ABB RAPID module: Module1.mod

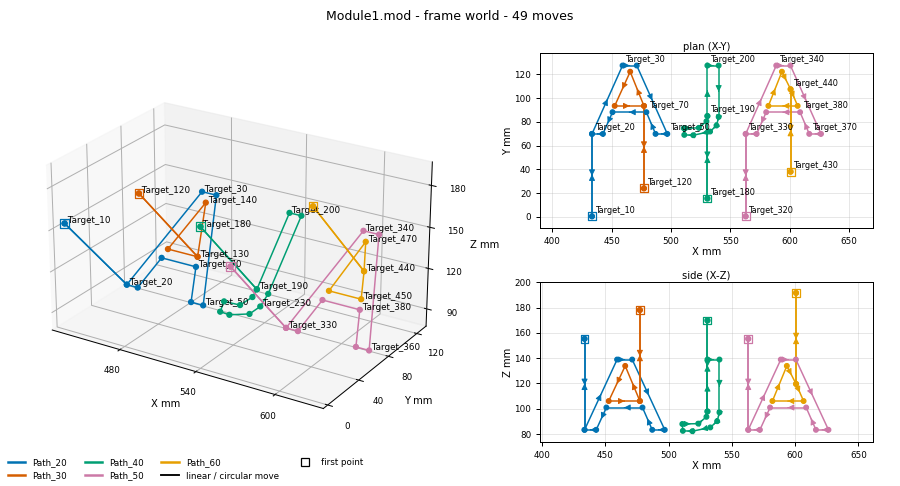
[picture p0: tool path of Module1.mod in frame world, 49 of 55 moves have a stored position in this frame; points joined in program order, loops and branches not executed]
MODULE Module1
        CONST robtarget Target_10:=[[-33.51704764,187.401145356,100.000301826],[0.00000002,-0.58897389,0.808152063,0.000000028],[-1,1,-1,1],[9E+09,9E+09,9E+09,9E+09,9E+09,9E+09]];
    CONST robtarget Target_20:=[[-33.51704764,187.401152167,0.000301826],[0.00000002,-0.58897389,0.808152063,0.000000028],[0,1,-1,1],[9E+09,9E+09,9E+09,9E+09,9E+09,9E+09]];
    CONST robtarget Target_30:=[[-59.250836036,107.401152167,0.000296377],[0.00000002,-0.58897389,0.808152063,0.000000028],[0,1,-1,1],[9E+09,9E+09,9E+09,9E+09,9E+09,9E+09]];
    CONST robtarget Target_40:=[[-71.196228528,107.401152167,0.000296377],[0.00000002,-0.58897389,0.808152063,0.000000028],[0,1,-1,1],[9E+09,9E+09,9E+09,9E+09,9E+09,9E+09]];
    CONST robtarget Target_50:=[[-96.930016924,187.401152167,0.000301826],[0.000000025,0.720360186,-0.693600175,-0.000000024],[0,1,-1,1],[9E+09,9E+09,9E+09,9E+09,9E+09,9E+09]];
    CONST robtarget Target_60:=[[-87.032406002,187.401152167,0.000301826],[0.00000002,-0.58897389,0.808152063,0.000000028],[0,1,-1,1],[9E+09,9E+09,9E+09,9E+09,9E+09,9E+09]];
    CONST robtarget Target_70:=[[-79.319095422,162.0086607,0.000300096],[0.00000002,-0.58897389,0.808152063,0.000000028],[0,1,-1,1],[9E+09,9E+09,9E+09,9E+09,9E+09,9E+09]];
    CONST robtarget Target_80:=[[-50.786672214,162.0086607,0.000300096],[0.00000002,-0.58897389,0.808152063,0.000000028],[0,1,-1,1],[9E+09,9E+09,9E+09,9E+09,9E+09,9E+09]];
    CONST robtarget Target_90:=[[-42.732064705,187.401152167,0.000301826],[0.00000002,-0.58897389,0.808152063,0.000000028],[0,1,-1,1],[9E+09,9E+09,9E+09,9E+09,9E+09,9E+09]];
    CONST robtarget Target_100:=[[-33.51704764,187.401152167,0.000301826],[0.00000002,-0.58897389,0.808152063,0.000000028],[0,1,-1,1],[9E+09,9E+09,9E+09,9E+09,9E+09,9E+09]];
    CONST robtarget Target_110:=[[-33.51704764,187.401145356,100.000301826],[0.00000002,-0.58897389,0.808152063,0.000000028],[-1,1,-1,1],[9E+09,9E+09,9E+09,9E+09,9E+09,9E+09]];
    CONST robtarget Target_120:=[[-77.271313852,154.636640237,100.000299594],[0.000000027,0.803729665,-0.594994644,-0.000000021],[0,1,-1,1],[9E+09,9E+09,9E+09,9E+09,9E+09,9E+09]];
    CONST robtarget Target_130:=[[-77.271313852,154.636647047,0.000299594],[-0.000000027,0.803729665,-0.594994644,-0.000000021],[0,1,-1,1],[9E+09,9E+09,9E+09,9E+09,9E+09,9E+09]];
    CONST robtarget Target_140:=[[-65.667218289,114.636647047,0.00029687],[-0.000000027,0.803729665,-0.594994644,-0.000000021],[0,1,-1,1],[9E+09,9E+09,9E+09,9E+09,9E+09,9E+09]];
    CONST robtarget Target_150:=[[-52.629675627,154.636647047,0.000299594],[-0.000000027,0.803729665,-0.594994644,-0.000000021],[0,1,-1,1],[9E+09,9E+09,9E+09,9E+09,9E+09,9E+09]];
    CONST robtarget Target_160:=[[-77.271313852,154.636647047,0.000299594],[-0.000000027,0.803729665,-0.594994644,-0.000000021],[0,1,-1,1],[9E+09,9E+09,9E+09,9E+09,9E+09,9E+09]];
    CONST robtarget Target_170:=[[-77.271313852,154.636640237,100.000299594],[-0.000000027,0.803729665,-0.594994644,-0.000000021],[0,1,-1,1],[9E+09,9E+09,9E+09,9E+09,9E+09,9E+09]];
    CONST robtarget Target_180:=[[-130.684278975,166.513773343,100.000300403],[-0.000000024,0.819152044,-0.573576437,-0.000000024],[0,1,-1,1],[9E+09,9E+09,9E+09,9E+09,9E+09,9E+09]];
    CONST robtarget Target_190:=[[-130.684278975,166.513780154,0.000300403],[0.000000024,-0.707106781,0.707106781,0.000000024],[0,1,-1,1],[9E+09,9E+09,9E+09,9E+09,9E+09,9E+09]];
    CONST robtarget Target_200:=[[-130.684278975,107.401152167,0.000296377],[0.000000024,-0.707106781,0.707106781,0.000000024],[0,1,-1,1],[9E+09,9E+09,9E+09,9E+09,9E+09,9E+09]];
    CONST robtarget Target_210:=[[-140.172333582,107.401152167,0.000296377],[0.000000024,-0.707106781,0.707106781,0.000000024],[0,1,-1,1],[9E+09,9E+09,9E+09,9E+09,9E+09,9E+09]];
    CONST robtarget Target_220:=[[-140.172333582,167.537670939,0.000300473],[0.000000024,0.819152044,-0.573576437,-0.000000024],[0,1,-1,1],[9E+09,9E+09,9E+09,9E+09,9E+09,9E+09]];
    CONST robtarget Target_230:=[[-138.363459862,177.588865478,0.000301158],[0.000000024,0.819152044,-0.573576437,-0.000000024],[0,1,-1,1],[9E+09,9E+09,9E+09,9E+09,9E+09,9E+09]];
    CONST robtarget Target_240:=[[-132.936838702,184.67077674,0.00030164],[0.000000024,0.819152044,-0.573576437,-0.000000024],[0,1,-1,1],[9E+09,9E+09,9E+09,9E+09,9E+09,9E+09]];
    CONST robtarget Target_250:=[[-118.807145869,188.971118037,0.000301932],[0.000000024,-0.707106781,0.707106781,0.000000024],[0,1,-1,1],[9E+09,9E+09,9E+09,9E+09,9E+09,9E+09]];
    CONST robtarget Target_260:=[[-111.23035406,188.561561724,0.000301905],[0.000000024,-0.707106781,0.707106781,0.000000024],[0,1,-1,1],[9E+09,9E+09,9E+09,9E+09,9E+09,9E+09]];
    CONST robtarget Target_270:=[[-110.820797746,180.779991758,0.000301375],[0.000000024,-0.707106781,0.707106781,0.000000024],[0,1,-1,1],[9E+09,9E+09,9E+09,9E+09,9E+09,9E+09]];
    CONST robtarget Target_280:=[[-123.482913787,180.353370597,0.000301346],[0.000000024,-0.707106781,0.707106781,0.000000024],[0,1,-1,1],[9E+09,9E+09,9E+09,9E+09,9E+09,9E+09]];
    CONST robtarget Target_290:=[[-129.882231193,172.605930324,0.000300819],[0.000000024,-0.707106781,0.707106781,0.000000024],[0,1,-1,1],[9E+09,9E+09,9E+09,9E+09,9E+09,9E+09]];
    CONST robtarget Target_300:=[[-130.684278975,166.513780154,0.000300403],[0.000000024,-0.707106781,0.707106781,0.000000024],[0,1,-1,1],[9E+09,9E+09,9E+09,9E+09,9E+09,9E+09]];
    CONST robtarget Target_310:=[[-130.684278975,166.513773343,100.000300403],[0.000000024,0.819152044,-0.573576437,-0.000000024],[0,1,-1,1],[9E+09,9E+09,9E+09,9E+09,9E+09,9E+09]];
    CONST robtarget Target_320:=[[-162.936835762,187.401145356,100.000301826],[-0.000000002,0.707106782,-0.70710678,-0.000000035],[-1,1,-1,1],[9E+09,9E+09,9E+09,9E+09,9E+09,9E+09]];
    CONST robtarget Target_330:=[[-162.936835762,187.401152167,0.000301826],[0.000000002,0.707106782,-0.70710678,-0.000000035],[0,1,-1,1],[9E+09,9E+09,9E+09,9E+09,9E+09,9E+09]];
    CONST robtarget Target_340:=[[-188.670624158,107.401152167,0.000296377],[0.000000002,0.707106782,-0.70710678,-0.000000035],[0,1,-1,1],[9E+09,9E+09,9E+09,9E+09,9E+09,9E+09]];
    CONST robtarget Target_350:=[[-200.61601665,107.401152167,0.000296377],[0.000000002,0.707106782,-0.70710678,-0.000000035],[0,1,-1,1],[9E+09,9E+09,9E+09,9E+09,9E+09,9E+09]];
    CONST robtarget Target_360:=[[-226.349805046,187.401152167,0.000301826],[0.000000002,0.707106782,-0.70710678,-0.000000035],[0,1,-1,1],[9E+09,9E+09,9E+09,9E+09,9E+09,9E+09]];
    CONST robtarget Target_370:=[[-216.452194124,187.401152167,0.000301826],[0.000000002,0.707106782,-0.70710678,-0.000000035],[0,1,-1,1],[9E+09,9E+09,9E+09,9E+09,9E+09,9E+09]];
    CONST robtarget Target_380:=[[-208.738883544,162.0086607,0.000300096],[0.000000002,0.707106782,-0.70710678,-0.000000035],[0,1,-1,1],[9E+09,9E+09,9E+09,9E+09,9E+09,9E+09]];
    CONST robtarget Target_390:=[[-180.206460336,162.0086607,0.000300096],[0.000000002,0.707106782,-0.70710678,-0.000000035],[0,1,-1,1],[9E+09,9E+09,9E+09,9E+09,9E+09,9E+09]];
    CONST robtarget Target_400:=[[-172.151852827,187.401152167,0.000301826],[0.000000002,0.707106782,-0.70710678,-0.000000035],[0,1,-1,1],[9E+09,9E+09,9E+09,9E+09,9E+09,9E+09]];
    CONST robtarget Target_410:=[[-162.936835762,187.401152167,0.000301826],[0.000000002,0.707106782,-0.70710678,-0.000000035],[0,1,-1,1],[9E+09,9E+09,9E+09,9E+09,9E+09,9E+09]];
    CONST robtarget Target_420:=[[-162.936835762,187.401145356,100.000301826],[0.000000002,0.707106782,-0.70710678,-0.000000035],[-1,1,-1,1],[9E+09,9E+09,9E+09,9E+09,9E+09,9E+09]];
    CONST robtarget Target_430:=[[-200.752535421,135.182715322,100.00029827],[0.000000021,-0.61876536,0.785575858,0.000000027],[0,1,-1,1],[9E+09,9E+09,9E+09,9E+09,9E+09,9E+09]];
    CONST robtarget Target_440:=[[-200.752535421,135.182722133,0.000298269],[0.000000021,-0.61876536,0.785575858,0.000000027],[0,1,-1,1],[9E+09,9E+09,9E+09,9E+09,9E+09,9E+09]];
    CONST robtarget Target_450:=[[-206.691101974,154.636647047,0.000299594],[0.000000021,-0.61876536,0.785575858,0.000000027],[0,1,-1,1],[9E+09,9E+09,9E+09,9E+09,9E+09,9E+09]];
    CONST robtarget Target_460:=[[-182.049463749,154.636647047,0.000299594],[0.000000021,-0.61876536,0.785575858,0.000000027],[0,1,-1,1],[9E+09,9E+09,9E+09,9E+09,9E+09,9E+09]];
    CONST robtarget Target_470:=[[-193.448781155,114.636647047,0.00029687],[0.000000021,-0.61876536,0.785575858,0.000000027],[0,1,-1,1],[9E+09,9E+09,9E+09,9E+09,9E+09,9E+09]];
    CONST robtarget Target_480:=[[-200.752535421,135.182722133,0.000298269],[0.000000021,-0.61876536,0.785575858,0.000000027],[0,1,-1,1],[9E+09,9E+09,9E+09,9E+09,9E+09,9E+09]];
    CONST robtarget Target_490:=[[-200.752535421,135.182715322,100.00029827],[0.000000021,-0.61876536,0.785575858,0.000000027],[0,1,-1,1],[9E+09,9E+09,9E+09,9E+09,9E+09,9E+09]];
    CONST jointtarget HomeP:=[[0,0,0,0,0,0],[9E+09,9E+09,9E+09,9E+09,9E+09,9E+09]];
    CONST jointtarget JointTarget_1:=[[0,20,-20,40,-20,-20],[9E+09,9E+09,9E+09,9E+09,9E+09,9E+09]];
    CONST jointtarget JointTarget_2:=[[0,50,-40,70,-50,-50],[9E+09,9E+09,9E+09,9E+09,9E+09,9E+09]];
!***********************************************************
    !
    ! Módulo:  Module1
    !
    ! Descripción:
    !   <Introduzca la descripción aquí>
    !
    ! Autor: equip
    !
    ! Versión: 1.0
    !
    !***********************************************************


    !***********************************************************
    !
    ! Procedimiento Main
    !
    !   Este es el punto de entrada de su programa
    !
    !***********************************************************
    PROC main()
        Security;
        Path_20;
        Path_30;
        Path_40;
        Path_50;
        Path_60;
        ToHome;
    ENDPROC
    PROC Path_20()
        MoveL Target_10,v50,z10,TCP1AJA\WObj:=WO1AJA;
        MoveL Target_20,v50,z10,TCP1AJA\WObj:=WO1AJA;
        MoveL Target_30,v50,z10,TCP1AJA\WObj:=WO1AJA;
        MoveL Target_40,v50,z10,TCP1AJA\WObj:=WO1AJA;
        MoveL Target_50,v50,z10,TCP1AJA\WObj:=WO1AJA;
        MoveL Target_60,v50,z10,TCP1AJA\WObj:=WO1AJA;
        MoveL Target_70,v50,z10,TCP1AJA\WObj:=WO1AJA;
        MoveL Target_80,v50,z10,TCP1AJA\WObj:=WO1AJA;
        MoveL Target_90,v50,z10,TCP1AJA\WObj:=WO1AJA;
        MoveL Target_100,v50,z10,TCP1AJA\WObj:=WO1AJA;
        MoveL Target_110,v50,z10,TCP1AJA\WObj:=WO1AJA;
    ENDPROC
    PROC Path_30()
        MoveL Target_120,v50,z10,TCP1AJA\WObj:=WO1AJA;
        MoveL Target_130,v50,z10,TCP1AJA\WObj:=WO1AJA;
        MoveL Target_140,v50,z10,TCP1AJA\WObj:=WO1AJA;
        MoveL Target_150,v50,z10,TCP1AJA\WObj:=WO1AJA;
        MoveL Target_160,v50,z10,TCP1AJA\WObj:=WO1AJA;
        MoveL Target_170,v50,z10,TCP1AJA\WObj:=WO1AJA;
    ENDPROC
    PROC Path_40()
        MoveL Target_180,v50,z10,TCP1AJA\WObj:=WO1AJA;
        MoveL Target_190,v50,z10,TCP1AJA\WObj:=WO1AJA;
        MoveL Target_200,v50,z10,TCP1AJA\WObj:=WO1AJA;
        MoveL Target_210,v50,z10,TCP1AJA\WObj:=WO1AJA;
        MoveL Target_220,v50,z10,TCP1AJA\WObj:=WO1AJA;
        MoveL Target_230,v50,z10,TCP1AJA\WObj:=WO1AJA;
        MoveL Target_240,v50,z10,TCP1AJA\WObj:=WO1AJA;
        MoveL Target_250,v50,z10,TCP1AJA\WObj:=WO1AJA;
        MoveL Target_260,v50,z10,TCP1AJA\WObj:=WO1AJA;
        MoveL Target_270,v50,z10,TCP1AJA\WObj:=WO1AJA;
        MoveL Target_280,v50,z10,TCP1AJA\WObj:=WO1AJA;
        MoveL Target_290,v50,z10,TCP1AJA\WObj:=WO1AJA;
        MoveL Target_300,v50,z10,TCP1AJA\WObj:=WO1AJA;
        MoveL Target_310,v50,z10,TCP1AJA\WObj:=WO1AJA;
    ENDPROC
    PROC Path_50()
        MoveL Target_320,v50,z10,TCP1AJA\WObj:=WO1AJA;
        MoveL Target_330,v50,z10,TCP1AJA\WObj:=WO1AJA;
        MoveL Target_340,v50,z10,TCP1AJA\WObj:=WO1AJA;
        MoveL Target_350,v50,z10,TCP1AJA\WObj:=WO1AJA;
        MoveL Target_360,v50,z10,TCP1AJA\WObj:=WO1AJA;
        MoveL Target_370,v50,z10,TCP1AJA\WObj:=WO1AJA;
        MoveL Target_380,v50,z10,TCP1AJA\WObj:=WO1AJA;
        MoveL Target_390,v50,z10,TCP1AJA\WObj:=WO1AJA;
        MoveL Target_400,v50,z10,TCP1AJA\WObj:=WO1AJA;
        MoveL Target_410,v50,z10,TCP1AJA\WObj:=WO1AJA;
        MoveL Target_420,v50,z10,TCP1AJA\WObj:=WO1AJA;
    ENDPROC
    PROC Path_60()
        MoveL Target_430,v50,z10,TCP1AJA\WObj:=WO1AJA;
        MoveL Target_440,v50,z10,TCP1AJA\WObj:=WO1AJA;
        MoveL Target_450,v50,z10,TCP1AJA\WObj:=WO1AJA;
        MoveL Target_460,v50,z10,TCP1AJA\WObj:=WO1AJA;
        MoveL Target_470,v50,z10,TCP1AJA\WObj:=WO1AJA;
        MoveL Target_480,v50,z10,TCP1AJA\WObj:=WO1AJA;
        MoveL Target_490,v50,z10,TCP1AJA\WObj:=WO1AJA;
    ENDPROC
    PROC Security()
        MoveAbsJ HomeP,v50,z10,TCP1AJA\WObj:=WO1AJA;
        MoveAbsJ JointTarget_1,v50,z10,TCP1AJA\WObj:=WO1AJA;
        MoveAbsJ JointTarget_2,v50,z10,TCP1AJA\WObj:=WO1AJA;
    ENDPROC
    PROC ToHome()
        MoveAbsJ JointTarget_2,v50,z10,TCP1AJA\WObj:=WO1AJA;
        MoveAbsJ JointTarget_1,v50,z10,TCP1AJA\WObj:=WO1AJA;
        MoveAbsJ HomeP,v50,z10,TCP1AJA\WObj:=WO1AJA;
    ENDPROC
ENDMODULE
